FUNCTION InitMotors: BOOL
VAR_INPUT
END_VAR
VAR
END_VAR

Automatic.MotorRot.ACPosition := 0;
Automatic.MotorRot.CurrentPosition := 0;
Automatic.MotorRot.Movement := FALSE;
Automatic.MotorRot.Direction := IO.MotorRotationDirection;

Automatic.MotorLif.ACPosition := 0;
Automatic.MotorLif.CurrentPosition := 0;
Automatic.MotorLif.Movement := FALSE;
Automatic.MotorLif.Direction := IO.MotorLiftingDirection;

Automatic.MotorExt.ACPosition := 0;
Automatic.MotorExt.CurrentPosition := 0;
Automatic.MotorExt.Movement := FALSE;
Automatic.MotorExt.Direction := IO.MotorExtensionDirection;

Automatic.MotorGri.ACPosition := 0;
Automatic.MotorGri.CurrentPosition := 0;
Automatic.MotorGri.Movement := FALSE;
Automatic.MotorGri.Direction := IO.MotorGripDirection;

END_FUNCTION

(* stored: Version 1.1.0.1, ProductVersion 3.1.4024.13
   POU InitMotors: Id {7fc36455-eee4-4b95-b6cf-e7b44cbc3396}, SpecialFunc None *)
